(* Logix 5000 project; controller corte_tubos Emulate 5570 rev 32.11; software revision 32.00 *)

TASK MainTask (continuous, watchdog 500 ms) : MainProgram

MODULES
   Local : Emulate 5570 (ICP 2, rev 32.11)
      I_O : vendor 1 type 0 code 15 (ICP 3, rev 1.1, Output RPI 50 ms)
END_MODULES

VAR_GLOBAL   (* controller tags *)
   Alarm : BOOL;
   Alarma : BOOL;
   apagar_alarma : BOOL;
   aprox_tubo_stop : SFC_STOP;
   cerrar_suj_fija_stop : SFC_STOP;
   Cerrar_suj_movil_stop : SFC_STOP;
   Config : BOOL;
   cont : DINT;
   cortar_stop : SFC_STOP;
   devolv_suj_movil_stop : SFC_STOP;
   dh : DINT;
   E : DINT;
   e1 : DINT;
   error : BOOL;
   K : ALIAS FOR Local:3:O.Data[0].0;
   long_tubo : DINT;
   n : DINT;
   off : DINT;
   POS_ALCANZADA : ALIAS FOR Local:3:I.Data[1].7;
   posicionar_tubo_stop : SFC_STOP;
   rdh : DINT;
   S1 : ALIAS FOR Local:3:I.Data[1].1;
   S2 : ALIAS FOR Local:3:I.Data[1].2;
   S3 : ALIAS FOR Local:3:I.Data[1].3;
   S4 : ALIAS FOR Local:3:I.Data[1].4;
   S5 : ALIAS FOR Local:3:I.Data[1].5;
   S6 : ALIAS FOR Local:3:I.Data[1].6;
   selector1 : DINT;
   Start : ALIAS FOR Local:3:I.Data[1].8;
   Step_100 : SFC_STEP := (Status := 16#0020_0000, PauseTimer := 1);
   Step_101 : SFC_STEP := (Status := 16#0020_0000, PauseTimer := 1);
   Step_200 : SFC_STEP := (Status := 16#0020_0000, PauseTimer := 1);
   Step_201 : SFC_STEP := (Status := 16#0020_0000, PauseTimer := 1);
   Step_202 : SFC_STEP := (Status := 16#0020_0000, PauseTimer := 1);
   Step_203 : SFC_STEP := (Status := 16#0020_0000, PauseTimer := 1, PRE := 500);
   Step_204 : SFC_STEP := (Status := 16#0020_0000, PauseTimer := 1);
   Step_205 : SFC_STEP := (Status := 16#0020_0000, PauseTimer := 1);
   Step_206 : SFC_STEP := (Status := 16#0020_0000, PauseTimer := 1);
   Step_207 : SFC_STEP := (Status := 16#0020_0000, PauseTimer := 1, PRE := 500);
   Step_208 : SFC_STEP := (Status := 16#0020_0000, PauseTimer := 1);
   Step_209 : SFC_STEP := (Status := 16#0020_0000, PauseTimer := 1);
   Step_210 : SFC_STEP := (Status := 16#0020_0000, PauseTimer := 1);
   Step_211 : SFC_STEP := (Status := 16#0020_0000, PauseTimer := 1);
   Step_300 : SFC_STEP := (Status := 16#0020_0000, PauseTimer := 1);
   Step_301 : SFC_STEP := (Status := 16#0020_0000, PauseTimer := 1);
   Step_302 : SFC_STEP := (Status := 16#0020_0000, PauseTimer := 1);
   Step_400 : SFC_STEP := (Status := 16#0020_0000, PauseTimer := 1);
   Step_401 : SFC_STEP := (Status := 16#0020_0000, PauseTimer := 1);
   Step_402 : SFC_STEP := (Status := 16#0020_0000, PauseTimer := 1);
   Step_403 : SFC_STEP := (Status := 16#0020_0000, PauseTimer := 1);
   Step_500 : SFC_STEP := (Status := 16#0020_0000, PauseTimer := 1);
   Step_501 : SFC_STEP := (Status := 16#0020_0000, PauseTimer := 1);
   Step_502 : SFC_STEP := (Status := 16#0020_0000, PauseTimer := 1, PRE := 200);
   Step_503 : SFC_STEP := (Status := 16#0020_0000, PauseTimer := 1);
   Step_504 : SFC_STEP := (Status := 16#0020_0000, PauseTimer := 1);
   Step_600 : SFC_STEP := (Status := 16#0020_0000, PauseTimer := 1);
   Step_601 : SFC_STEP := (Status := 16#0020_0000, PauseTimer := 1);
   Step_602 : SFC_STEP := (Status := 16#0020_0000, PauseTimer := 1);
   Step_700 : SFC_STEP := (Status := 16#0020_0000, PauseTimer := 1);
   Stop : ALIAS FOR Local:3:I.Data[1].9;
   tipo_tubo : DINT;
   Tran_005 : BOOL;
   Y1 : ALIAS FOR Local:3:O.Data[0].1;
   Y2 : ALIAS FOR Local:3:O.Data[0].2;
   Y3 : ALIAS FOR Local:3:O.Data[0].3;
   Y4 : ALIAS FOR Local:3:O.Data[0].4;
   Y5 : ALIAS FOR Local:3:O.Data[0].5;
   Y6 : ALIAS FOR Local:3:O.Data[0].6;
END_VAR

PROGRAM MainProgram   (* main routine MainRoutine *)
VAR
   Action_000 : SFC_ACTION := (Status := 16#0020_0000, PauseTimer := 1);
   Action_001 : SFC_ACTION := (Status := 16#0020_0000, PauseTimer := 1);
   Action_002 : SFC_ACTION := (Status := 16#0020_0000, PauseTimer := 1);
   Action_003 : SFC_ACTION := (Status := 16#0020_0000, PauseTimer := 1);
   Action_004 : SFC_ACTION := (Status := 16#0020_0000, PauseTimer := 1);
   Action_005 : SFC_ACTION := (Status := 16#0020_0000, PauseTimer := 1);
   Action_006 : SFC_ACTION := (Status := 16#0020_0000, PauseTimer := 1);
   Action_007 : SFC_ACTION := (Status := 16#0020_0000, PauseTimer := 1);
   Action_008 : SFC_ACTION := (Status := 16#0020_0000, PauseTimer := 1);
   Action_009 : SFC_ACTION := (Status := 16#0020_0000, PauseTimer := 1);
   Action_010 : SFC_ACTION := (Status := 16#0020_0000, PauseTimer := 1);
   Action_011 : SFC_ACTION := (Status := 16#0020_0000, PauseTimer := 1);
   Action_012 : SFC_ACTION := (Status := 16#0020_0000, PauseTimer := 1);
   Action_013 : SFC_ACTION := (Status := 16#0020_0000, PauseTimer := 1);
   Action_014 : SFC_ACTION := (Status := 16#0020_0000, PauseTimer := 1);
   Action_015 : SFC_ACTION := (Status := 16#0020_0000, PauseTimer := 1);
   Action_016 : SFC_ACTION := (Status := 16#0020_0000, PauseTimer := 1);
   Action_017 : SFC_ACTION := (Status := 16#0020_0000, PauseTimer := 1);
   Action_018 : SFC_ACTION := (Status := 16#0020_0000, PauseTimer := 1);
   Action_019 : SFC_ACTION := (Status := 16#0020_0000, PauseTimer := 1);
   Action_020 : SFC_ACTION := (Status := 16#0020_0000, PauseTimer := 1);
   Action_021 : SFC_ACTION := (Status := 16#0020_0000, PauseTimer := 1);
   Action_022 : SFC_ACTION := (Status := 16#0020_0000, PauseTimer := 1);
   Action_023 : SFC_ACTION := (Status := 16#0020_0000, PauseTimer := 1);
   Action_024 : SFC_ACTION := (Status := 16#0020_0000, PauseTimer := 1);
   Action_025 : SFC_ACTION := (Status := 16#0020_0000, PauseTimer := 1);
   Action_026 : SFC_ACTION := (Status := 16#0020_0000, PauseTimer := 1);
   Action_027 : SFC_ACTION := (Status := 16#0020_0000, PauseTimer := 1);
   Action_028 : SFC_ACTION := (Status := 16#0020_0000, PauseTimer := 1);
   Action_029 : SFC_ACTION := (Status := 16#0020_0000, PauseTimer := 1);
   Action_030 : SFC_ACTION := (Status := 16#0020_0000, PauseTimer := 1);
   Action_031 : SFC_ACTION := (Status := 16#0020_0000, PauseTimer := 1);
   Action_032 : SFC_ACTION := (Status := 16#0020_0000, PauseTimer := 1);
   Action_033 : SFC_ACTION := (Status := 16#0020_0000, PauseTimer := 1);
   Action_034 : SFC_ACTION := (Status := 16#0020_0000, PauseTimer := 1);
   Action_035 : SFC_ACTION := (Status := 16#0020_0000, PauseTimer := 1);
   Action_036 : SFC_ACTION := (Status := 16#0020_0000, PauseTimer := 1);
   Step_000 : SFC_STEP := (Status := 16#0020_0000, PauseTimer := 1);
   Step_001 : SFC_STEP := (Status := 16#0020_0000, PauseTimer := 1);
   Step_002 : SFC_STEP := (Status := 16#0020_0000, PauseTimer := 1);
   Step_003 : SFC_STEP := (Status := 16#0020_0000, PauseTimer := 1);
   Step_004 : SFC_STEP := (Status := 16#0020_0000, PauseTimer := 1, PRE := 2000);
   Step_005 : SFC_STEP := (Status := 16#0020_0000, PauseTimer := 1);
   Step_006 : SFC_STEP := (Status := 16#0020_0000, PauseTimer := 1);
   Step_007 : SFC_STEP := (Status := 16#0020_0000, PauseTimer := 1);
   Step_008 : SFC_STEP := (Status := 16#0020_0000, PauseTimer := 1);
   Step_009 : SFC_STEP := (Status := 16#0020_0000, PauseTimer := 1);
   Step_010 : SFC_STEP := (Status := 16#0020_0000, PauseTimer := 1);
   Step_011 : SFC_STEP := (Status := 16#0020_0000, PauseTimer := 1);
   Step_012 : SFC_STEP := (Status := 16#0020_0000, PauseTimer := 1);
   Step_013 : SFC_STEP := (Status := 16#0020_0000, PauseTimer := 1);
   Step_014 : SFC_STEP := (Status := 16#0020_0000, PauseTimer := 1);
   Step_015 : SFC_STEP := (Status := 16#0020_0000, PauseTimer := 1);
   Step_016 : SFC_STEP := (Status := 16#0020_0000, PauseTimer := 1);
   Step_017 : SFC_STEP := (Status := 16#0020_0000, PauseTimer := 1);
   Step_018 : SFC_STEP := (Status := 16#0020_0000, PauseTimer := 1);
   Step_019 : SFC_STEP := (Status := 16#0020_0000, PauseTimer := 1);
   Step_020 : SFC_STEP := (Status := 16#0020_0000, PauseTimer := 1);
   Step_021 : SFC_STEP := (Status := 16#0020_0000, PauseTimer := 1);
   Step_022 : SFC_STEP := (Status := 16#0020_0000, PauseTimer := 1);
   Step_023 : SFC_STEP := (Status := 16#0020_0000, PauseTimer := 1);
   Step_024 : SFC_STEP := (Status := 16#0020_0000, PauseTimer := 1);
   Step_025 : SFC_STEP := (Status := 16#0020_0000, PauseTimer := 1);
   Step_026 : SFC_STEP := (Status := 16#0020_0000, PauseTimer := 1);
   Step_027 : SFC_STEP := (Status := 16#0020_0000, PauseTimer := 1);
   Step_028 : SFC_STEP := (Status := 16#0020_0000, PauseTimer := 1);
   Step_029 : SFC_STEP := (Status := 16#0020_0000, PauseTimer := 1);
   Step_030 : SFC_STEP := (Status := 16#0020_0000, PauseTimer := 1);
   Step_031 : SFC_STEP := (Status := 16#0020_0000, PauseTimer := 1);
   Step_032 : SFC_STEP := (Status := 16#0020_0000, PauseTimer := 1);
   Step_033 : SFC_STEP := (Status := 16#0020_0000, PauseTimer := 1);
   Step_034 : SFC_STEP := (Status := 16#0020_0000, PauseTimer := 1);
   Step_035 : SFC_STEP := (Status := 16#0020_0000, PauseTimer := 1);
   Step_036 : SFC_STEP := (Status := 16#0020_0000, PauseTimer := 1);
   Step_037 : SFC_STEP := (Status := 16#0020_0000, PauseTimer := 1);
   Step_038 : SFC_STEP := (Status := 16#0020_0000, PauseTimer := 1);
   Step_039 : SFC_STEP := (Status := 16#0020_0000, PauseTimer := 1);
   Step_040 : SFC_STEP := (Status := 16#0020_0000, PauseTimer := 1);
   Stop_000 : SFC_STOP;
   Stop_001 : SFC_STOP;
   Stop_002 : SFC_STOP;
   Stop_003 : SFC_STOP;
   Stop_004 : SFC_STOP;
   Stop_005 : SFC_STOP;
   Tran_000 : BOOL;
   Tran_001 : BOOL;
   Tran_002 : BOOL;
   Tran_003 : BOOL;
   Tran_004 : BOOL;
   Tran_007 : BOOL;
   Tran_008 : BOOL;
   Tran_009 : BOOL;
   Tran_010 : BOOL;
   Tran_011 : BOOL;
   Tran_013 : BOOL;
   Tran_015 : BOOL;
   Tran_017 : BOOL;
   Tran_019 : BOOL;
   Tran_021 : BOOL;
   Tran_022 : BOOL;
   Tran_023 : BOOL;
   Tran_025 : BOOL;
   Tran_026 : BOOL;
   Tran_029 : BOOL;
   Tran_030 : BOOL;
   Tran_032 : BOOL;
   Tran_033 : BOOL;
   Tran_034 : BOOL;
   Tran_035 : BOOL;
   Tran_036 : BOOL;
   Tran_037 : BOOL;
   Tran_039 : BOOL;
   Tran_041 : BOOL;
   Tran_042 : BOOL;
   Tran_043 : BOOL;
   Tran_044 : BOOL;
END_VAR

ROUTINE aproximar_tubo   (* sequential function chart *)
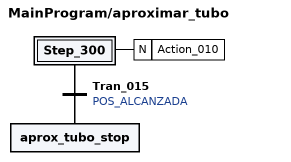
   INITIAL_STEP Step_300:
      ACTION Action_010 (N):
         rdh:=off;
      END_ACTION
   END_STEP
   TRANSITION Tran_015 FROM Step_300 TO aprox_tubo_stop
      := POS_ALCANZADA
   END_TRANSITION
   STOP aprox_tubo_stop;
END_ROUTINE

ROUTINE calcular_parametros   (* structured text *)
   case tipo_tubo OF
   	1: long_tubo:=115;
   	2: long_tubo:=540;
   	3: long_tubo:=600;
   	4: long_tubo:=69;
   	5: long_tubo:=200;
   	6: long_tubo:=430;
   	7: long_tubo:=430;
   	8: long_tubo:=450;
   	9: long_tubo:=950;
   	10: long_tubo:=950;
   	11: long_tubo:=400;
   	12: long_tubo:=400;
   end_case;
   if NOT long_tubo = 0 then
   	error:=1;
   else
   	error:=0;
   end_if;
   n:=6000/long_tubo;
   off:=50;
END_ROUTINE

ROUTINE cerrar_suj_fija   (* sequential function chart *)
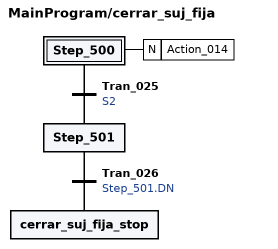
   INITIAL_STEP Step_500:
      ACTION Action_014 (N):
         Y2[:=]1;
      END_ACTION
   END_STEP
   TRANSITION Tran_025 FROM Step_500 TO Step_501
      := S2
   END_TRANSITION
   STEP Step_501:
   END_STEP
   TRANSITION Tran_026 FROM Step_501 TO cerrar_suj_fija_stop
      := Step_501.DN
   END_TRANSITION
   STOP cerrar_suj_fija_stop;
END_ROUTINE

ROUTINE cerrar_suj_movil   (* sequential function chart *)
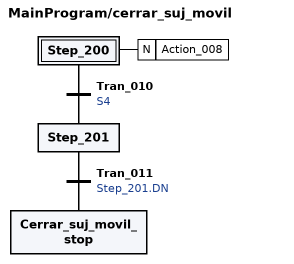
   INITIAL_STEP Step_200:
      ACTION Action_008 (N):
         Y4[:=]1;
      END_ACTION
   END_STEP
   TRANSITION Tran_010 FROM Step_200 TO Step_201
      := S4
   END_TRANSITION
   STEP Step_201:
   END_STEP
   TRANSITION Tran_011 FROM Step_201 TO Cerrar_suj_movil_stop
      := Step_201.DN
   END_TRANSITION
   STOP Cerrar_suj_movil_stop;
END_ROUTINE

ROUTINE config_inicial   (* structured text *)
   Y1:=1;
   Y2:=0;
   Y3:=1;
   Y4:=0;
   Y5:=1;
   Y6:=0;
   rdh:=0;
   K:=0;
   cont:=1;
END_ROUTINE

ROUTINE cortar   (* sequential function chart *)
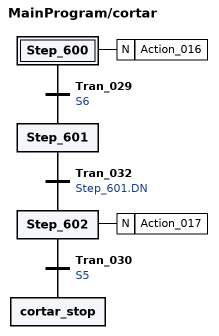
   INITIAL_STEP Step_600:
      ACTION Action_016 (N):
         Y6[:=]1;
      END_ACTION
   END_STEP
   TRANSITION Tran_029 FROM Step_600 TO Step_601
      := S6
   END_TRANSITION
   STEP Step_601:
   END_STEP
   TRANSITION Tran_032 FROM Step_601 TO Step_602
      := Step_601.DN
   END_TRANSITION
   STEP Step_602:
      ACTION Action_017 (N):
         Y5[:=]1;
      END_ACTION
   END_STEP
   TRANSITION Tran_030 FROM Step_602 TO cortar_stop
      := S5
   END_TRANSITION
   STOP cortar_stop;
END_ROUTINE

ROUTINE devolver_suj_movil   (* sequential function chart *)
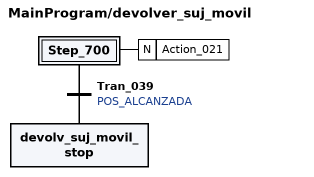
   INITIAL_STEP Step_700:
      ACTION Action_021 (N):
         rdh:=off;
      END_ACTION
   END_STEP
   TRANSITION Tran_039 FROM Step_700 TO devolv_suj_movil_stop
      := POS_ALCANZADA
   END_TRANSITION
   STOP devolv_suj_movil_stop;
END_ROUTINE

ROUTINE Grafcet_general   (* sequential function chart *)
// secuencia de corte general
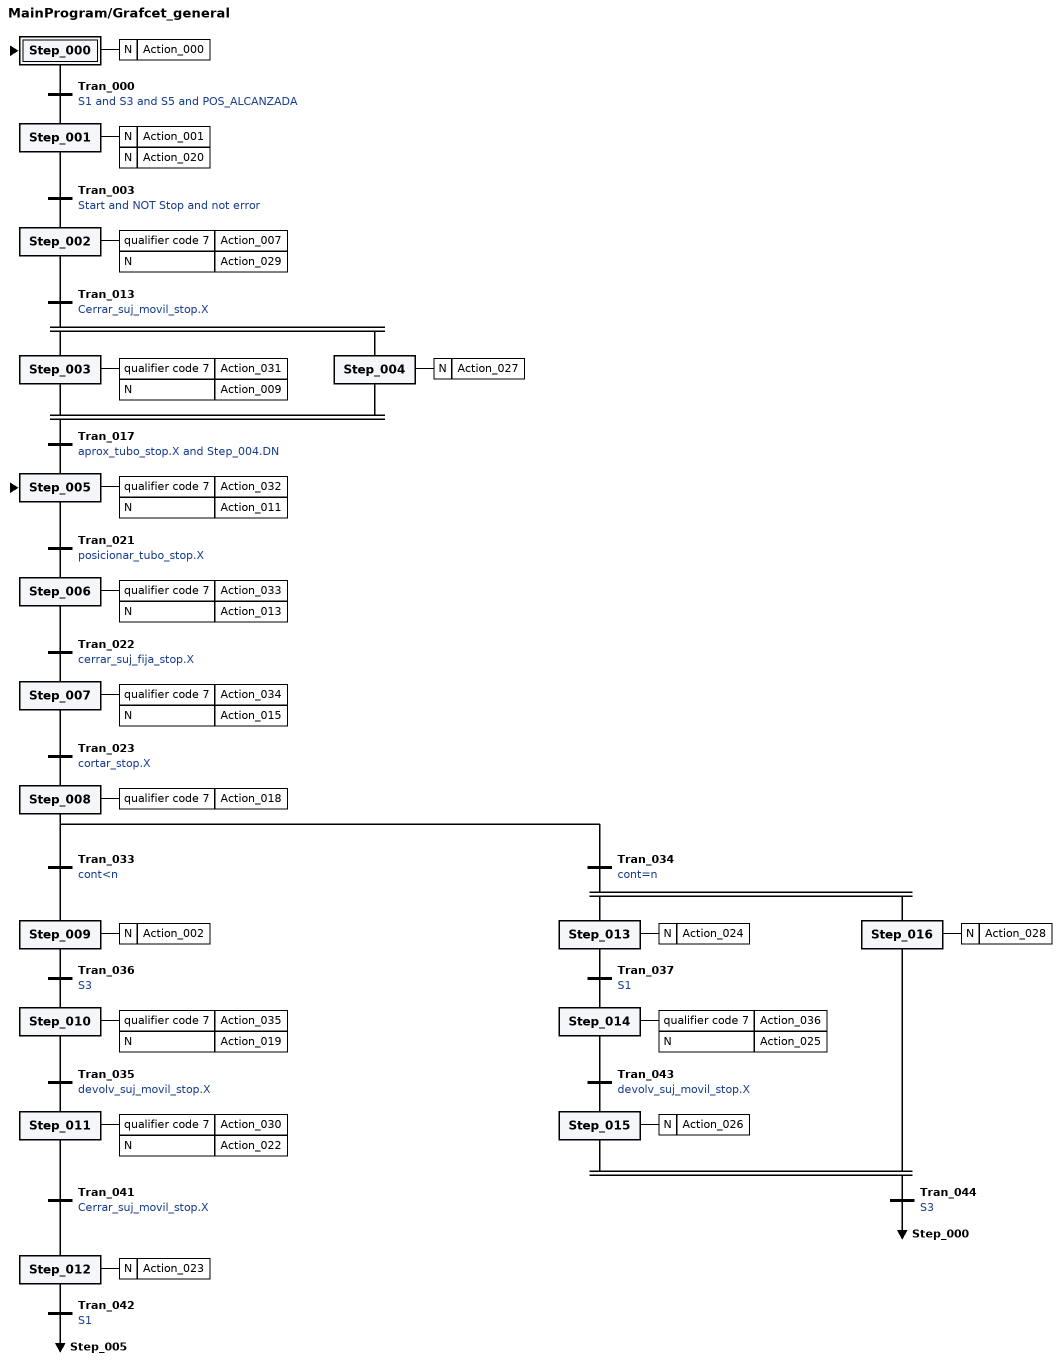
   INITIAL_STEP Step_000:
      ACTION Action_000 (N):
         JSR(config_inicial);
      END_ACTION
   END_STEP
   TRANSITION Tran_000 FROM Step_000 TO Step_001
      := S1 and S3 and S5 and POS_ALCANZADA
   END_TRANSITION
   STEP Step_001:
      ACTION Action_001 (N):
         Y1:=0;
         Y3:=0;
         Y5:=0;
      END_ACTION
      ACTION Action_020 (N):
         JSR(calcular_parametros);
      END_ACTION
   END_STEP
   TRANSITION Tran_003 FROM Step_001 TO Step_002
      := Start and NOT Stop and not error
   END_TRANSITION
   STEP Step_002:
      ACTION Action_007 (qualifier code 7):
         SFR(cerrar_suj_movil,Step_200);
         Cerrar_suj_movil_stop.X:=0;
      END_ACTION
      ACTION Action_029 (N):
         JSR(cerrar_suj_movil);
      END_ACTION
   END_STEP
   TRANSITION Tran_013 FROM Step_002 TO (Step_003, Step_004)
      := Cerrar_suj_movil_stop.X
   END_TRANSITION
   STEP Step_003:
      ACTION Action_031 (qualifier code 7):
         SFR(aproximar_tubo,Step_300);
         aprox_tubo_stop.X:=0;
      END_ACTION
      ACTION Action_009 (N):
         JSR(aproximar_tubo);
      END_ACTION
   END_STEP
   STEP Step_004:
      ACTION Action_027 (N):
         K:=1;
      END_ACTION
   END_STEP
   TRANSITION Tran_017 FROM (Step_003, Step_004) TO Step_005
      := aprox_tubo_stop.X and Step_004.DN
   END_TRANSITION
   STEP Step_005:
      ACTION Action_032 (qualifier code 7):
         SFR(posicionar_tubo,Step_400);
         posicionar_tubo_stop.X:=0;
      END_ACTION
      ACTION Action_011 (N):
         JSR(posicionar_tubo);
      END_ACTION
   END_STEP
   TRANSITION Tran_021 FROM Step_005 TO Step_006
      := posicionar_tubo_stop.X
   END_TRANSITION
   STEP Step_006:
      ACTION Action_033 (qualifier code 7):
         SFR(cerrar_suj_fija,Step_500);
         cerrar_suj_fija_stop.X:=0;
      END_ACTION
      ACTION Action_013 (N):
         JSR(cerrar_suj_fija);
      END_ACTION
   END_STEP
   TRANSITION Tran_022 FROM Step_006 TO Step_007
      := cerrar_suj_fija_stop.X
   END_TRANSITION
   STEP Step_007:
      ACTION Action_034 (qualifier code 7):
         SFR(cortar,Step_600);
         cortar_stop.X:=0;
      END_ACTION
      ACTION Action_015 (N):
         JSR(cortar);
      END_ACTION
   END_STEP
   TRANSITION Tran_023 FROM Step_007 TO Step_008
      := cortar_stop.X
   END_TRANSITION
   STEP Step_008:
      ACTION Action_018 (qualifier code 7):
         cont:=cont+1;
      END_ACTION
   END_STEP
   TRANSITION Tran_033 FROM Step_008 TO Step_009
      := cont<n
   END_TRANSITION
   TRANSITION Tran_034 FROM Step_008 TO (Step_013, Step_016)
      := cont=n
   END_TRANSITION
   STEP Step_009:
      ACTION Action_002 (N):
         Y3[:=]1;
      END_ACTION
   END_STEP
   TRANSITION Tran_036 FROM Step_009 TO Step_010
      := S3
   END_TRANSITION
   STEP Step_013:
      ACTION Action_024 (N):
         Y1[:=]1;
      END_ACTION
   END_STEP
   STEP Step_010:
      ACTION Action_035 (qualifier code 7):
         SFR(devolver_suj_movil,Step_700);
         devolv_suj_movil_stop.X:=0;
      END_ACTION
      ACTION Action_019 (N):
         JSR(devolver_suj_movil);
      END_ACTION
   END_STEP
   TRANSITION Tran_037 FROM Step_013 TO Step_014
      := S1
   END_TRANSITION
   STEP Step_016:
      ACTION Action_028 (N):
         K:=0;
      END_ACTION
   END_STEP
   STEP Step_014:
      ACTION Action_036 (qualifier code 7):
         SFR(devolver_suj_movil,Step_700);
         devolv_suj_movil_stop.X:=0;
      END_ACTION
      ACTION Action_025 (N):
         JSR(devolver_suj_movil);
      END_ACTION
   END_STEP
   TRANSITION Tran_035 FROM Step_010 TO Step_011
      := devolv_suj_movil_stop.X
   END_TRANSITION
   TRANSITION Tran_043 FROM Step_014 TO Step_015
      := devolv_suj_movil_stop.X
   END_TRANSITION
   STEP Step_011:
      ACTION Action_030 (qualifier code 7):
         SFR(cerrar_suj_movil,Step_200);
         Cerrar_suj_movil_stop.X:=0;
      END_ACTION
      ACTION Action_022 (N):
         JSR(cerrar_suj_movil);
      END_ACTION
   END_STEP
   TRANSITION Tran_041 FROM Step_011 TO Step_012
      := Cerrar_suj_movil_stop.X
   END_TRANSITION
   STEP Step_015:
      ACTION Action_026 (N):
         Y3[:=]1;
      END_ACTION
   END_STEP
   STEP Step_012:
      ACTION Action_023 (N):
         Y1[:=]1;
      END_ACTION
   END_STEP
   TRANSITION Tran_044 FROM (Step_015, Step_016) TO Step_000
      := S3
   END_TRANSITION
   TRANSITION Tran_042 FROM Step_012 TO Step_005
      := S1
   END_TRANSITION
END_ROUTINE

ROUTINE MainRoutine   (* ladder *)
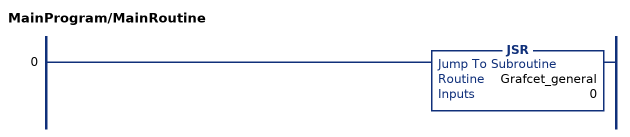
   0: JSR(Grafcet_general,0);
END_ROUTINE

ROUTINE posicionar_tubo   (* sequential function chart *)
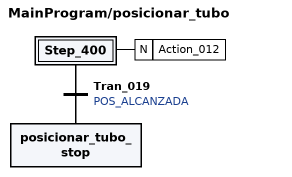
   INITIAL_STEP Step_400:
      ACTION Action_012 (N):
         rdh:=off+long_tubo;
      END_ACTION
   END_STEP
   TRANSITION Tran_019 FROM Step_400 TO posicionar_tubo_stop
      := POS_ALCANZADA
   END_TRANSITION
   STOP posicionar_tubo_stop;
END_ROUTINE
END_PROGRAM
